FUNCTION Convert_TIME_TO_DATE : Hresult
VAR_INPUT
	in : TIME;
	out : REFERENCE TO DATE;
END_VAR
VAR
	converted : DATE;
END_VAR
VAR CONSTANT
	INCOMPATIBLE : HRESULT := 16#9811070E;
END_VAR

converted := TIME_TO_DATE(in);

IF (DATE_TO_TIME(converted) <> in) THEN
	Convert_TIME_TO_DATE := INCOMPATIBLE;
	RETURN;
END_IF

out := converted;

END_FUNCTION

(* stored: Version 1.1.0.1, ProductVersion 3.1.4024.12
   POU Convert_TIME_TO_DATE: Id {1c16f169-aa10-4dbe-8aab-cb8087a0e2f1}, SpecialFunc None *)
